(* CODESYS project TP_INF_IND_RENAN_JULIA.project

Project tree, tasks and I/O mapping:
  Device : CODESYS Control Win V3, 3S - Smart Software Solutions GmbH, order no. 305021, version 3.5.11.40
    application Application
      libraries: Standard, * (System)
      task MainTask (cyclic, interval t#20ms, priority 1) calls Main
      task Simulacao (cyclic, interval t#20ms, priority 1) calls Simulacao
      task Controle (cyclic, interval t#20ms, priority 1) calls Controle
      program Main [ST]
      pou Simulacao [ST]
      pou Controle [ST]
*)

// Device/Application/Main
PROGRAM Main
VAR_INPUT
    (* Entradas dos Sensores *)
    Vagao_Posicionado: BOOL;
    Peso_Silo1: REAL;
    Peso_Silo2: REAL;
    Nivel_Baixo_Silo1: BOOL;
    Nivel_Alto_Silo1: BOOL;
    Nivel_Baixo_Silo2: BOOL;
    Nivel_Alto_Silo2: BOOL;
    Caminhao_Posicionado: BOOL;
    Sensor_Presenca_Vagao: BOOL;
    Sensor_Presenca_Caminhao: BOOL;

    (* Comandos do SCADA *)
    Comando_Iniciar_Descarregamento: BOOL;
    Comando_Iniciar_Carregamento: BOOL;
    Capacidade_Caminhao: REAL;
    Modo_Manual: BOOL;
END_VAR

VAR_OUTPUT
    (* Estados e Monitoramento para o SCADA *)
    Estado_Descarregamento: INT;
    Estado_Carregamento: INT;
    Transportador_Entrada_ON: BOOL;
    Ventilacao_Silo1_ON: BOOL;
    Ventilacao_Silo2_ON: BOOL;
    Alimentador_Saida_ON: BOOL;
    Transportador_Saida_ON: BOOL;
    Alimentador_Moega1_ON: BOOL;
    Alimentador_Moega2_ON: BOOL;
    Moega_Pesagem_ON: BOOL;
    Desviador_Mangueira_POS: INT;
    Alarme_Transportador_IN: BOOL;
    Alarme_Transportador_OUT: BOOL;
    Alarme_Alimentador_OUT: BOOL;
    Alarme_Moega: BOOL;

    (* Feedback dos Sensores *)
    Feedback_Vagao_Posicionado: BOOL;
    Feedback_Peso_Silo1: REAL;
    Feedback_Peso_Silo2: REAL;
    Feedback_Nivel_Baixo_Silo1: BOOL;
    Feedback_Nivel_Alto_Silo1: BOOL;
    Feedback_Nivel_Baixo_Silo2: BOOL;
    Feedback_Nivel_Alto_Silo2: BOOL;
    Feedback_Caminhao_Posicionado: BOOL;
    Feedback_Sensor_Presenca_Vagao: BOOL;
    Feedback_Sensor_Presenca_Caminhao: BOOL;
END_VAR

VAR
    (* Variáveis Internas *)
    Interna_Descarregamento: INT := 0;
    Interna_Carregamento: INT := 0;
END_VAR

* Atualiza os feedbacks dos sensores para o SCADA *)
Feedback_Vagao_Posicionado := Vagao_Posicionado;
Feedback_Peso_Silo1 := Peso_Silo1;
Feedback_Peso_Silo2 := Peso_Silo2;
Feedback_Nivel_Baixo_Silo1 := Nivel_Baixo_Silo1;
Feedback_Nivel_Alto_Silo1 := Nivel_Alto_Silo1;
Feedback_Nivel_Baixo_Silo2 := Nivel_Baixo_Silo2;
Feedback_Nivel_Alto_Silo2 := Nivel_Alto_Silo2;
Feedback_Caminhao_Posicionado := Caminhao_Posicionado;
Feedback_Sensor_Presenca_Vagao := Sensor_Presenca_Vagao;
Feedback_Sensor_Presenca_Caminhao := Sensor_Presenca_Caminhao;

(* Chama a POU Controle *)
Controle(
    Vagao_Posicionado := Vagao_Posicionado,
    Peso_Silo1 := Peso_Silo1,
    Peso_Silo2 := Peso_Silo2,
    Nivel_Baixo_Silo1 := Nivel_Baixo_Silo1,
    Nivel_Alto_Silo1 := Nivel_Alto_Silo1,
    Nivel_Baixo_Silo2 := Nivel_Baixo_Silo2,
    Nivel_Alto_Silo2 := Nivel_Alto_Silo2,
    Caminhao_Posicionado := Caminhao_Posicionado,
    Sensor_Presenca_Vagao := Sensor_Presenca_Vagao,
    Sensor_Presenca_Caminhao := Sensor_Presenca_Caminhao,
    Comando_Iniciar_Descarregamento := Comando_Iniciar_Descarregamento,
    Comando_Iniciar_Carregamento := Comando_Iniciar_Carregamento,
    Capacidade_Caminhao := Capacidade_Caminhao,
    Modo_Manual := Modo_Manual,
    Estado_Descarregamento => Estado_Descarregamento,
    Estado_Carregamento => Estado_Carregamento,
    Transportador_Entrada_Ligado => Transportador_Entrada_Ligado,
    Ventilacao_Silo1_Ligada => Ventilacao_Silo1_Ligada,
    Ventilacao_Silo2_Ligada => Ventilacao_Silo2_Ligada,
    Alimentador_Saida_Ligado => Alimentador_Saida_Ligado,
    Transportador_Saida_Ligado => Transportador_Saida_Ligado,
    Alimentador_Moega1_Ligado => Alimentador_Moega1_Ligado,
    Alimentador_Moega2_Ligado => Alimentador_Moega2_Ligado,
    Moega_Pesagem_Ligada => Moega_Pesagem_Ligada,
    Desviador_Mangueira_Posicao => Desviador_Mangueira_Posicao,
    Alarme_Transportador_Entrada => Alarme_Transportador_Entrada,
    Alarme_Transportador_Saida => Alarme_Transportador_Saida,
    Alarme_Alimentador_Saida => Alarme_Alimentador_Saida,
    Alarme_Moega => Alarme_Moega,
    Interna_Descarregamento => Interna_Descarregamento,
    Interna_Carregamento => Interna_Carregamento
);

END_PROGRAM
